PROGRAM MC_State_MC
VAR
END_VAR

// NETWORK 1

END_PROGRAM

(* stored: Version 1.1.0.1, ProductVersion 3.1.4024.0
   POU MC_State_MC: Id {07cfa895-a264-45c1-986e-b77a48f71878}, SpecialFunc None *)
